TYPE ST_PML_Cmd :
STRUCT
    Cmd         : E_PML_Command;
    SeqId       : UDINT;     // increments each new command
END_STRUCT
END_TYPE

(* stored: Version 1.1.0.1, ProductVersion 3.1.4024.13
   DUT ST_PML_Cmd: Id {17c5ffbc-2472-4ff4-b8a1-d7fa549a932d} *)
